// TIA Portal V17 export
// export: Created 2024-09-02T12:49:54.5995138Z, ExportSetting WithDefaults, DisplayName Totally Integrated Automation Portal, DisplayVersion V17, DisplayName TIA Portal Openness, DisplayVersion V17, DisplayName TIA Portal Version Control Interface, DisplayVersion V17, DisplayName STEP 7 Professional, DisplayVersion V17, DisplayName STEP 7 Safety, DisplayVersion V17, DisplayName WinCC Professional, DisplayVersion V17
FUNCTION "AnwFC_ZP_Initialisation" : Void   // FC1, LAD
TITLE = Initialization / Initialisierung
{ S7_Optimized_Access := 'TRUE' }
AUTHOR : OlegFuehrus
FAMILY : AF
NAME : AF
VERSION : 1.0
// stored: AutoNumber false, IsIECCheckEnabled false, SetENOAutomatically false, UDAEnableTagReadback false
BEGIN

REGION Network 1: Initialization HMI System - OP70 / Initalisierung HMI System OP40
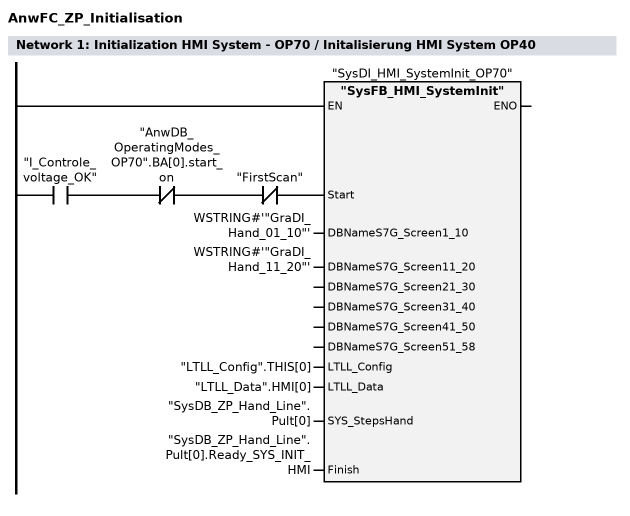
   RUNG wire#powerrail
      "SysDI_HMI_SystemInit_OP70"(Start := wire#w1, DBNameS7G_Screen1_10 := WSTRING#'"GraDI_Hand_01_10"', DBNameS7G_Screen11_20 := WSTRING#'"GraDI_Hand_11_20"', DBNameS7G_Screen21_30 :=, DBNameS7G_Screen31_40 :=, DBNameS7G_Screen41_50 :=, DBNameS7G_Screen51_58 :=, LTLL_Config := "LTLL_Config".THIS[0], LTLL_Data := "LTLL_Data".HMI[0], SYS_StepsHand := "SysDB_ZP_Hand_Line".Pult[0], Finish := "SysDB_ZP_Hand_Line".Pult[0].Ready_SYS_INIT_HMI)
   END_RUNG
   RUNG wire#powerrail
      Contact( "I_Controle_voltage_OK" )
      I_Contact( "AnwDB_OperatingModes_OP70".BA[0].start_on )
      I_Contact( "FirstScan" )
   END_RUNG wire#w1
   // the same network as SCL:
   "SysDI_HMI_SystemInit_OP70"(Start := "I_Controle_voltage_OK" AND NOT "AnwDB_OperatingModes_OP70".BA[0].start_on AND NOT "FirstScan",   // "SysFB_HMI_SystemInit"
                           DBNameS7G_Screen1_10 := WSTRING#'"GraDI_Hand_01_10"',
                           DBNameS7G_Screen11_20 := WSTRING#'"GraDI_Hand_11_20"',
                           LTLL_Config := "LTLL_Config".THIS[0],
                           LTLL_Data := "LTLL_Data".HMI[0],
                           SYS_StepsHand := "SysDB_ZP_Hand_Line".Pult[0],
                           Finish := "SysDB_ZP_Hand_Line".Pult[0].Ready_SYS_INIT_HMI);
END_REGION
END_FUNCTION
